Staubli VAL3: getByteAt.pgx

public program getByteAt(num x_nByteIndex, num& x_nBuffer[], num& x_nRes)
begin

  //Header begin

  // This function is trivial, it just return in "x_nRes" the "x_nByteIndex" element of the array x_nBuffer (most likely a plc's memory area you read with readArea()).
  //
  //Input parameters
  //
  // num x_nByteIndex: the index of the element in the "x_nBuffer[]" array representing the byte we want to read
	// num x_nBuffer[1]: the monodimensional array of num from where we are reading a byte.

  //Output parameters
  //
  // num x_nRes: where the result is stored

  //Examples
  //
  // 	call getByteAt(12, nDB, l_nRes)
  //
  //History
  // Creation: 24-12-16 - Alessio Villa
  //Header end

  x_nRes=x_nBuffer[x_nByteIndex]

end
